% RSLogix 500 project BLUE_BANNER_RESTACKER_JAN_14_2022_3_11PMPM_BAK013.RSS, saved by version 11.00.00.00 %
PROJECT "UNTITLED"    % processor: MicroLogix 1400 %

PROGRAM FILES
  LAD 2   34 rungs

DATA FILES
  O0 OUTPUT  6 elements
  I1 INPUT  8 elements
  S2 STATUS  66 elements
  B3 BINARY  2 elements
  T4 TIMER  6 elements
  C5 COUNTER  1 elements
  R6 CONTROL  1 elements
  N7 INTEGER  3 elements
  F8 FLOAT  1 elements

LADDER 2
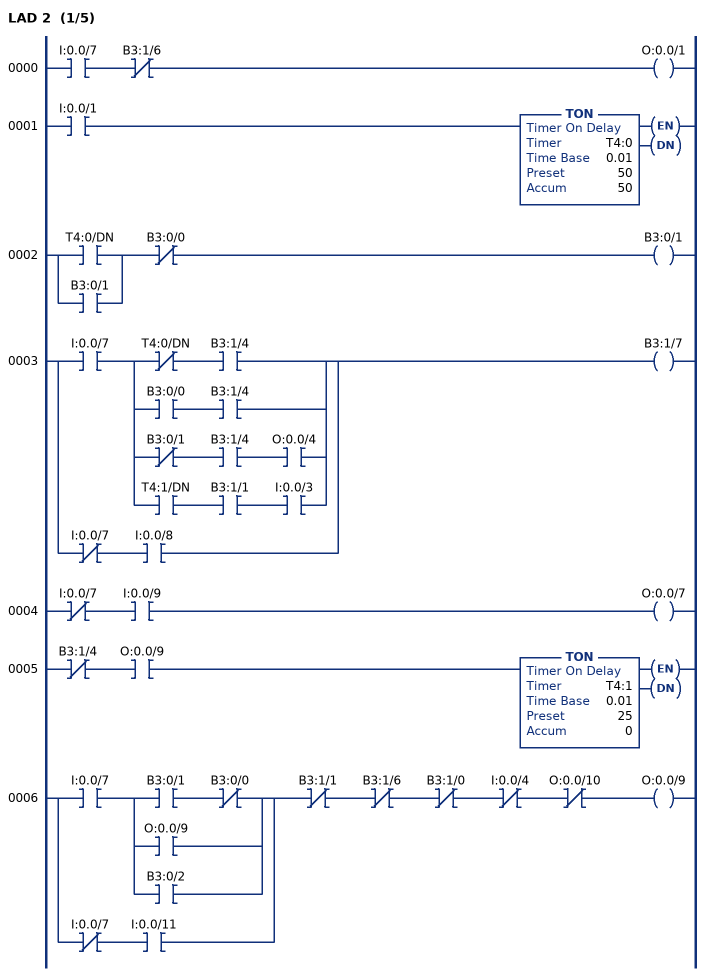
% Rung: 0 %
SOR XIC I:0.0/7 XIO B3:1/6 OTE O:0.0/1 EOR
% Rung: 1 %
SOR XIC I:0.0/1 TON T4:0 0.01 50 50 EOR
% Rung: 2 %
SOR BST XIC T4:0/DN NXB XIC B3:0/1 BND XIO B3:0/0 OTE B3:0/1 EOR
% Rung: 3 %
SOR BST XIC I:0.0/7 BST XIO T4:0/DN XIC B3:1/4 NXB BST XIC B3:0/0 XIC B3:1/4 NXB BST XIO B3:0/1 XIC B3:1/4 XIC O:0.0/4 NXB XIC T4:1/DN XIC B3:1/1 XIC I:0.0/3 BND BND BND NXB XIO I:0.0/7 XIC I:0.0/8 BND OTE B3:1/7 EOR
% Rung: 4 %
SOR XIO I:0.0/7 XIC I:0.0/9 OTE O:0.0/7 EOR
% Rung: 5 %
SOR XIO B3:1/4 XIC O:0.0/9 TON T4:1 0.01 25 0 EOR
% Rung: 6 %
SOR BST XIC I:0.0/7 BST XIC B3:0/1 XIO B3:0/0 NXB BST XIC O:0.0/9 NXB XIC B3:0/2 BND BND NXB XIO I:0.0/7 XIC I:0.0/11 BND XIO B3:1/1 XIO B3:1/6 XIO B3:1/0 XIO I:0.0/4 XIO O:0.0/10 OTE O:0.0/9 EOR

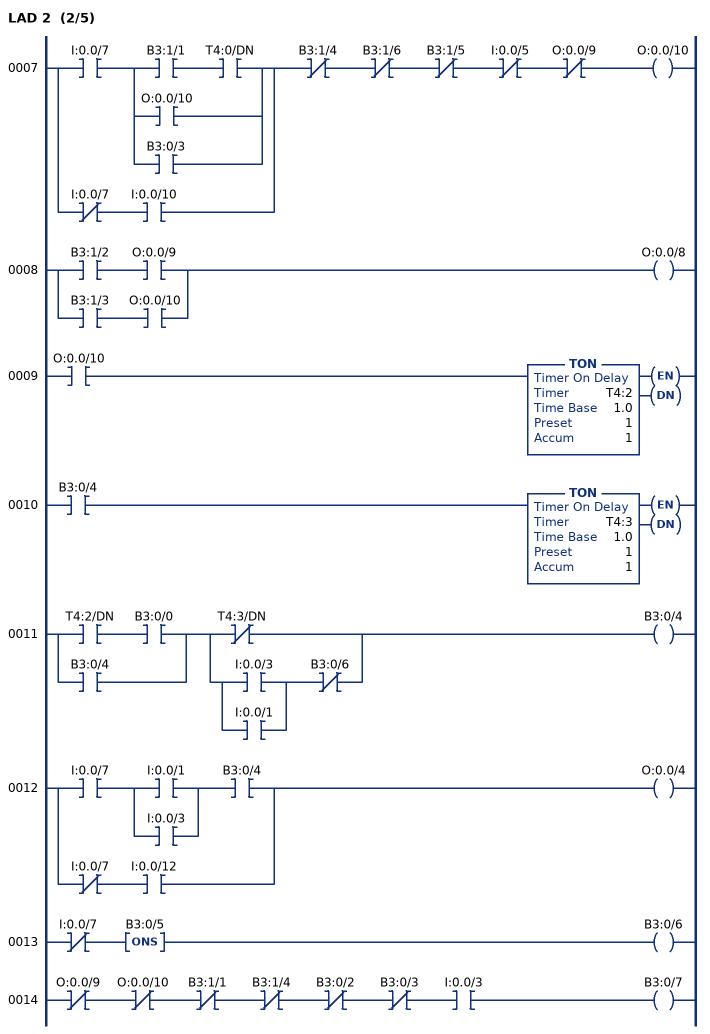
% Rung: 7 %
SOR BST XIC I:0.0/7 BST XIC B3:1/1 XIC T4:0/DN NXB BST XIC O:0.0/10 NXB XIC B3:0/3 BND BND NXB XIO I:0.0/7 XIC I:0.0/10 BND XIO B3:1/4 XIO B3:1/6 XIO B3:1/5 XIO I:0.0/5 XIO O:0.0/9 OTE O:0.0/10 EOR
% Rung: 8 %
SOR BST XIC B3:1/2 XIC O:0.0/9 NXB XIC B3:1/3 XIC O:0.0/10 BND OTE O:0.0/8 EOR
% Rung: 9 %
SOR XIC O:0.0/10 TON T4:2 1.0 1 1 EOR
% Rung: 10 %
SOR XIC B3:0/4 TON T4:3 1.0 1 1 EOR
% Rung: 11 %
SOR BST XIC T4:2/DN XIC B3:0/0 NXB XIC B3:0/4 BND BST XIO T4:3/DN NXB BST XIC I:0.0/3 NXB XIC I:0.0/1 BND XIO B3:0/6 BND OTE B3:0/4 EOR
% Rung: 12 %
SOR BST XIC I:0.0/7 BST XIC I:0.0/1 NXB XIC I:0.0/3 BND XIC B3:0/4 NXB XIO I:0.0/7 XIC I:0.0/12 BND OTE O:0.0/4 EOR
% Rung: 13 %
SOR XIO I:0.0/7 ONS B3:0/5 OTE B3:0/6 EOR
% Rung: 14 %
SOR XIO O:0.0/9 XIO O:0.0/10 XIO B3:1/1 XIO B3:1/4 XIO B3:0/2 XIO B3:0/3 XIC I:0.0/3 OTE B3:0/7 EOR

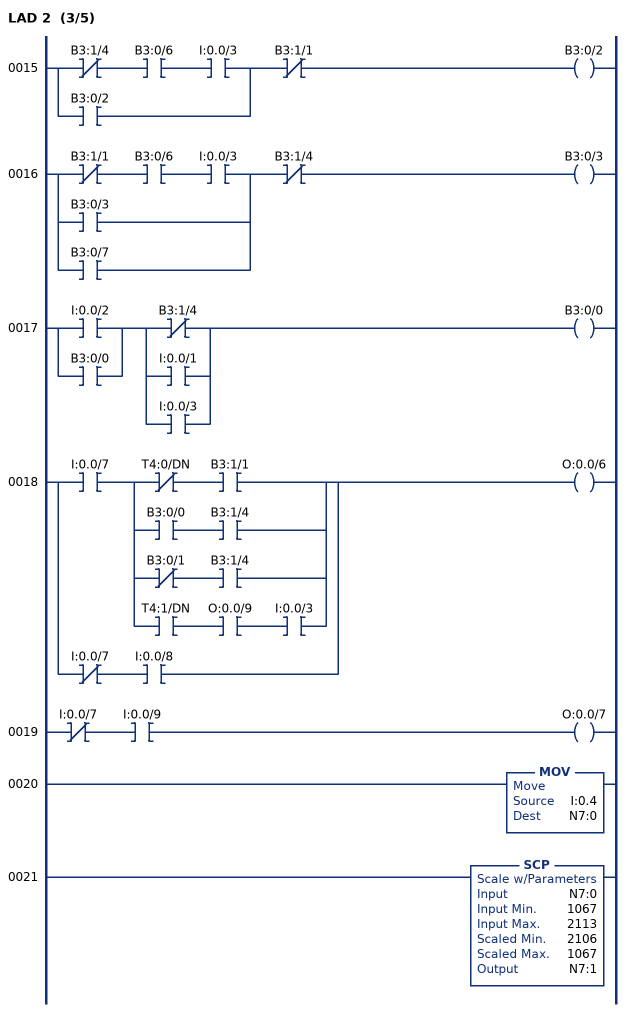
% Rung: 15 %
SOR BST XIO B3:1/4 XIC B3:0/6 XIC I:0.0/3 NXB XIC B3:0/2 BND XIO B3:1/1 OTE B3:0/2 EOR
% Rung: 16 %
SOR BST XIO B3:1/1 XIC B3:0/6 XIC I:0.0/3 NXB BST XIC B3:0/3 NXB XIC B3:0/7 BND BND XIO B3:1/4 OTE B3:0/3 EOR
% Rung: 17 %
SOR BST XIC I:0.0/2 NXB XIC B3:0/0 BND BST XIO B3:1/4 NXB BST XIC I:0.0/1 NXB XIC I:0.0/3 BND BND OTE B3:0/0 EOR
% Rung: 18 %
SOR BST XIC I:0.0/7 BST XIO T4:0/DN XIC B3:1/1 NXB BST XIC B3:0/0 XIC B3:1/4 NXB BST XIO B3:0/1 XIC B3:1/4 NXB XIC T4:1/DN XIC O:0.0/9 XIC I:0.0/3 BND BND BND NXB XIO I:0.0/7 XIC I:0.0/8 BND OTE O:0.0/6 EOR
% Rung: 19 %
SOR XIO I:0.0/7 XIC I:0.0/9 OTE O:0.0/7 EOR
% Rung: 20 %
SOR MOV I:0.4 N7:0 EOR
% Rung: 21 %
SOR SCP N7:0 1067 2113 2106 1067 N7:1 EOR

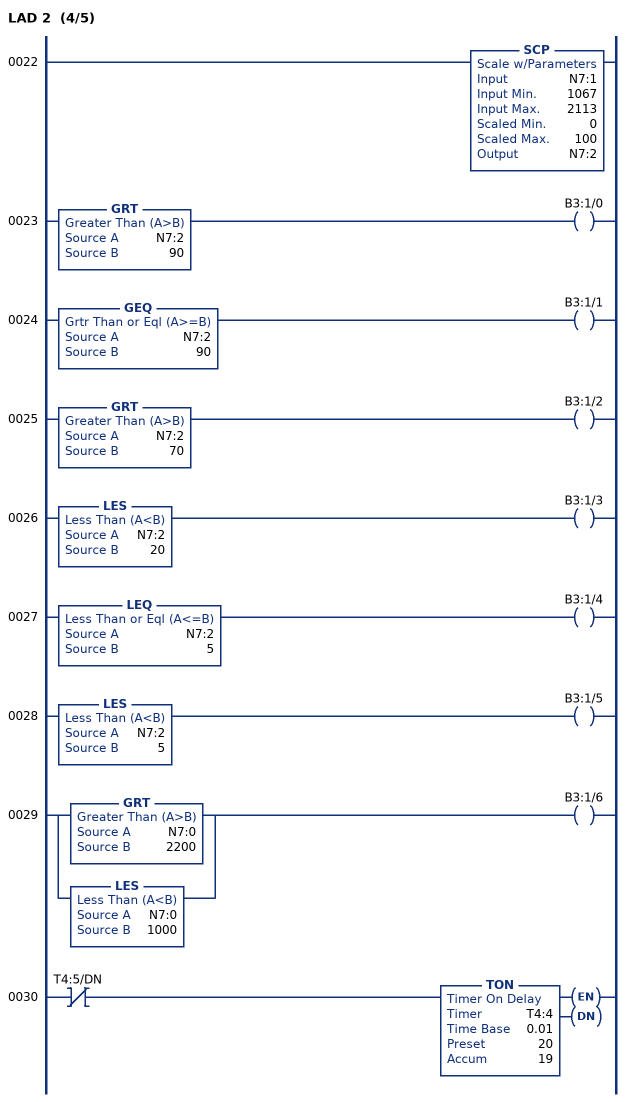
% Rung: 22 %
SOR SCP N7:1 1067 2113 0 100 N7:2 EOR
% Rung: 23 %
SOR GRT N7:2 90 OTE B3:1/0 EOR
% Rung: 24 %
SOR GEQ N7:2 90 OTE B3:1/1 EOR
% Rung: 25 %
SOR GRT N7:2 70 OTE B3:1/2 EOR
% Rung: 26 %
SOR LES N7:2 20 OTE B3:1/3 EOR
% Rung: 27 %  % edit flag set %
SOR LEQ N7:2 5 OTE B3:1/4 EOR
% Rung: 28 %  % edit flag set %
SOR LES N7:2 5 OTE B3:1/5 EOR
% Rung: 29 %
SOR BST GRT N7:0 2200 NXB LES N7:0 1000 BND OTE B3:1/6 EOR
% Rung: 30 %
SOR XIO T4:5/DN TON T4:4 0.01 20 19 EOR

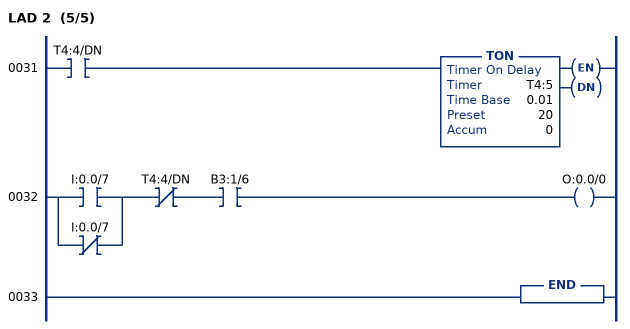
% Rung: 31 %
SOR XIC T4:4/DN TON T4:5 0.01 20 0 EOR
% Rung: 32 %
SOR BST XIC I:0.0/7 NXB XIO I:0.0/7 BND XIO T4:4/DN XIC B3:1/6 OTE O:0.0/0 EOR
% Rung: 33 %
SOR END EOR

REVISION NOTES
  0: stacker would not stack 4 bins, only up to 3. new encoder installed. Alan/Eulises.
  1: rung 25 edited: source B changed from 90 to 80. This should slow down the stacker going up sooner so that it does not hit the frame.
  2: Rung 25: 90 to 80. slow doen going up sooner to avoid hitting frame
  3: trying to use the 2hp VFD instead of the 7.5hp

DATA TABLE (non-zero values as saved)
DATA B3
% B3:0 % 0X0011 0X0038
DATA T4
% .PRE .ACC %
% T4:0 % 50 50
% T4:1 % 25 0
% T4:2 % 1 1
% T4:3 % 1 1
% T4:4 % 20 19
% T4:5 % 20 0
DATA N7
% N7:0 % 2118 1800 0
